ABB RAPID module: MainModule.modx

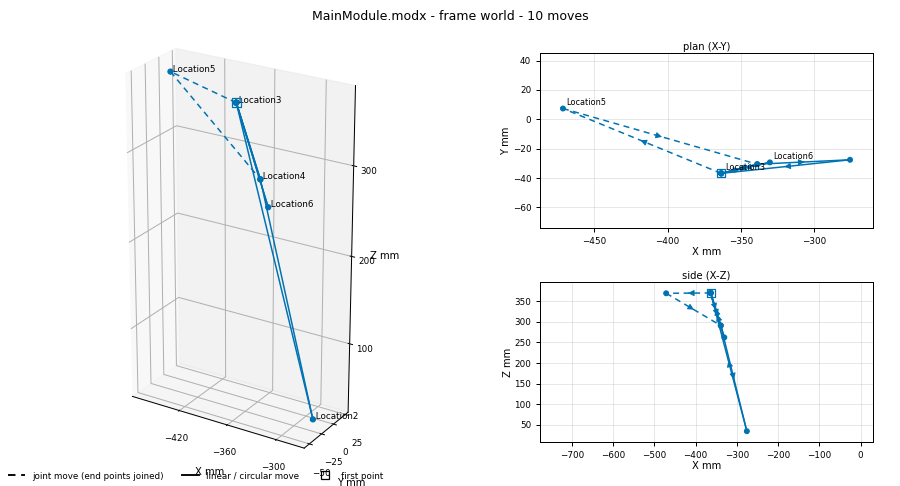
[picture p0: tool path of MainModule.modx in frame world, 10 of 10 moves have a stored position in this frame; points joined in program order, loops and branches not executed]
MODULE MainModule
CONST robtarget Target_20:=[[200, 200, 400], [0, 1, 0, 0], [1, 0, 0, 0], [145.7014269, 9000000000, 9000000000, 9000000000, 9000000000, 9000000000]];
CONST robtarget Target_30:=[[-200, 200, 400], [0, 1, 0, 0], [2, 0, 0, 0], [-102.158258441, 9000000000, 9000000000, 9000000000, 9000000000, 9000000000]];
PERS robtarget Location1:=[[-386.532745361328, -19.6524963378906, 315.689575195313], [0.204580903053284, 0.518802106380463, -0.775684237480164, -0.295474231243134], [-1, 0, 2, 0], [-95.209699574118, 9000000000, 9000000000, 9000000000, 9000000000, 9000000000]];
PERS robtarget Location2:=[[-275.788177490234, -27.5446434020996, 34.9423027038574], [0.074581973254681, -0.719046533107758, 0.690936803817749, -0.00399923883378506], [0, 0, 2, 4], [-83.9946711797192, 9000000000, 9000000000, 9000000000, 9000000000, 9000000000]];
PERS robtarget Location3:=[[-363.520629882813, -36.7881278991699, 369.898681640625], [0.00965851917862892, 0.693030714988708, -0.719793617725372, -0.0388873107731342], [0, 0, 1, 4], [-84.5925469522824, 9000000000, 9000000000, 9000000000, 9000000000, 9000000000]];
PERS robtarget Location4:=[[-338.966156005859, -30.5506534576416, 290.98779296875], [0.0456151217222214, -0.701731085777283, 0.710955679416656, 0.00589575851336122], [0, 0, 1, 4], [-85.20789003443, 9000000000, 9000000000, 9000000000, 9000000000, 9000000000]];
PERS robtarget Location5:=[[-471.236480712891, 7.36933422088623, 369.0986328125], [0.66135436296463, -0.288175493478775, -0.119181491434574, 0.682173788547516], [0, -2, 1, 4], [-82.9501356333978, 9000000000, 9000000000, 9000000000, 9000000000, 9000000000]];
PERS robtarget Location6:=[[-330.35693359375, -29.300802230835, 262.121856689453], [0.0478060767054558, -0.703067302703857, 0.709493935108185, 0.00541345169767737], [0, 0, 1, 4], [-85.4257072926204, 9000000000, 9000000000, 9000000000, 9000000000, 9000000000]];

CONST speeddata testSpeed:=v200;
PERS jointtarget calib_pos:=[[90,0,0,0,0,0],[0,9E+09,9E+09,9E+09,9E+09,9E+09]];
PROC main()
MoveJ Location3, v200, fine, wi_tGripper;
WaitTime 2;
MotionSup \On \TuneValue:= 50;

MoveJ Location3, v500, fine, wi_tGripper;
MoveL Location4, v50, fine, wi_tGripper;
MoveL Location3, v500, fine, wi_tGripper;
MotionSup \Off;
MoveL Location6, v1000, fine, wi_tGripper;
MotionSup \On \TuneValue:= 50;
MoveL Location3, v200, fine, wi_tGripper;
MoveJ Location5, v200, fine, wi_tGripper;
WaitTime 3;
MoveJ Location4, v200, fine, wi_tGripper;
MoveL Location2, v200, fine, wi_tGripper;
g_GripOut;
g_Stop;
MoveL Location3, v200, fine, wi_tGripper;
ENDPROC
ENDMODULE
